// TIA Portal V17 export
// export: Created 2024-08-09T12:53:14.3489012Z, ExportSetting WithDefaults, DisplayName Totally Integrated Automation Portal, DisplayVersion V17 Update 7, DisplayName TIA Portal Openness, DisplayVersion V17 Update 7, DisplayName TIA Portal Version Control Interface, DisplayVersion V17, DisplayName STEP 7 Professional, DisplayVersion V17 Update 7, DisplayName STEP 7 Safety, DisplayVersion V17 Update 6, DisplayName WinCC Professional, DisplayVersion V17 Update 7
VAR_GLOBAL   // PLC tag table "CIRCUIT EXPEDITION"
END_VAR
VAR_GLOBAL CONSTANT   // user constants
   NIV_CIR_EXP_DEBUT_LOT : USInt := 1;
   NIV_CIR_EXP_LANCE : USInt := 10;
   NIV_CIR_EXP_PRET : USInt := 20;
   NIV_CIR_EXP_VIDANGE : USInt := 30;
   NIV_CIR_EXP_FIN_LOT : USInt := 255;
END_VAR
